(* Visualisation GAS_CALIBRATION
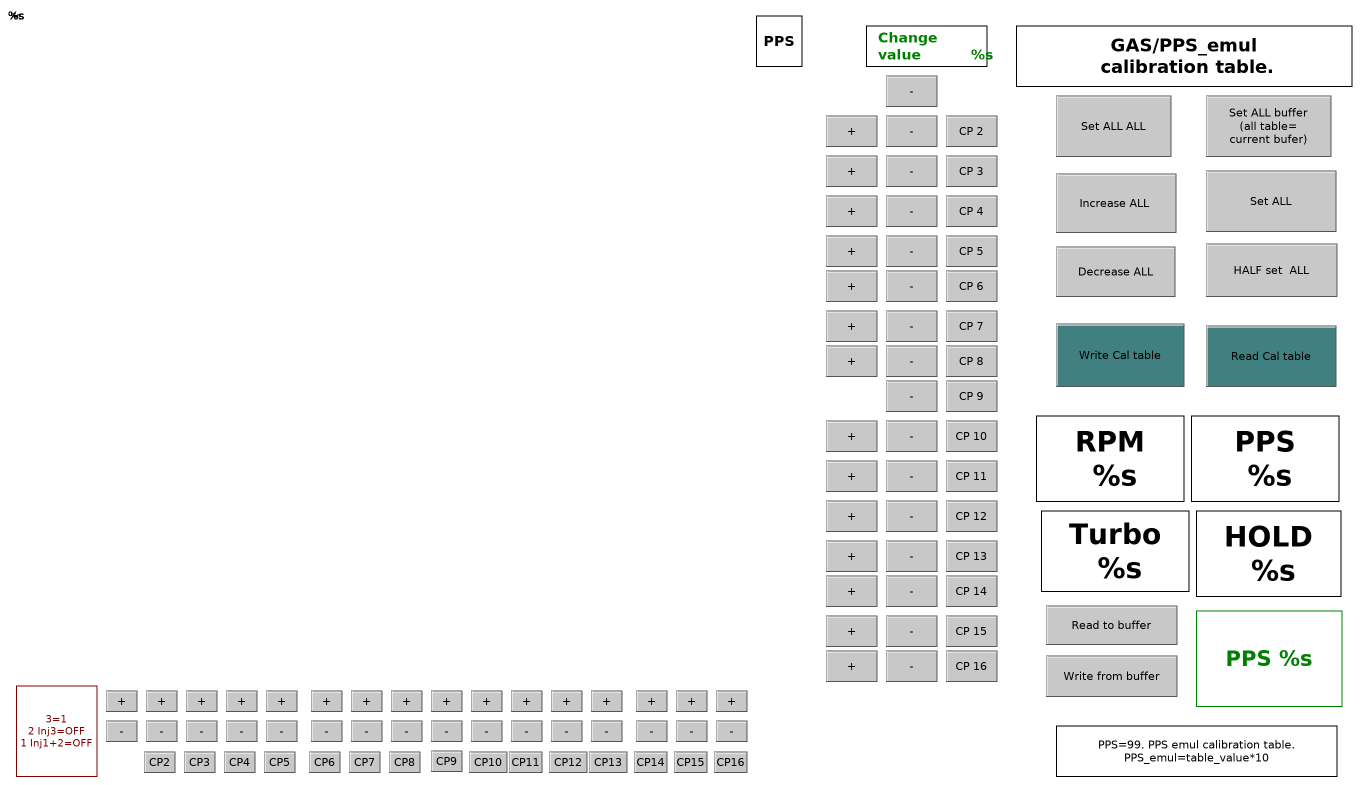
rectangle at (0,0)-(0,0): text "%s"; shows p.RPM_table[INDEX]; editable
rectangle at (0,0)-(0,0): text "%s"; shows p.Turbo_table[1]; editable
rectangle at (0,0)-(0,0): text "%s"; shows p.Turbo_table[2]; editable
rectangle at (0,0)-(0,0): text "%s"; shows p.Turbo_table[3]; editable
rectangle at (0,0)-(0,0): text "%s"; shows p.Turbo_table[4]; editable
rectangle at (0,0)-(0,0): text "%s"; shows p.Turbo_table[5]; editable
rectangle at (0,0)-(0,0): text "%s"; shows p.Turbo_table[6]; editable
rectangle at (0,0)-(0,0): text "%s"; shows p.Turbo_table[7]; editable
rectangle at (0,0)-(0,0): text "%s"; shows p.Turbo_table[8]; editable
rectangle at (0,0)-(0,0): text "%s"; shows p.Turbo_table[9]; editable
rectangle at (0,0)-(0,0): text "%s"; shows p.Turbo_table[10]; editable
rectangle at (0,0)-(0,0): text "%s"; shows p.Turbo_table[11]; editable
rectangle at (0,0)-(0,0): text "%s"; shows p.Turbo_table[12]; editable
rectangle at (0,0)-(0,0): text "%s"; shows p.Turbo_table[13]; editable
rectangle at (0,0)-(0,0): text "%s"; shows p.Turbo_table[14]; editable
rectangle at (0,0)-(0,0): text "%s"; shows p.Turbo_table[15]; editable
rectangle at (0,0)-(0,0): text "%s"; shows p.Turbo_table[16]; editable
rounded rectangle at (1180,595)-(1326,691): text "PPS %s"; shows DFPRS_Change_Cal_Table.PPS_number; editable
button at (1040,158)-(1160,217): text "Increase ALL"; taps DFPRS_Change_Cal_Table.ALL_plus
button at (1040,231)-(1159,281): text "Decrease ALL"; taps DFPRS_Change_Cal_Table.ALL_minus
button at (1190,310)-(1320,371): text "Read Cal table"; taps DFPRS_Change_Cal_Table.Read_cal
button at (1040,308)-(1168,371): text "Write Cal table"; taps DFPRS_Change_Cal_Table.Write_cal
button at (1190,155)-(1320,216): text "Set ALL"; taps DFPRS_Change_Cal_Table.Set_ALL
button at (1190,228)-(1321,281): text "HALF set  ALL"; taps DFPRS_Change_Cal_Table.HALF_set_ALL
button at (870,60)-(921,91): text "-"; taps DFPRS_Change_Cal_Table.RPM_Flag_minus_1
button at (810,100)-(861,131): text "+"; taps DFPRS_Change_Cal_Table.RPM_Flag_plus_2
button at (870,100)-(921,131): text "-"; taps DFPRS_Change_Cal_Table.RPM_Flag_minus_2
button at (930,100)-(981,131): text "CP 2"; taps DFPRS_Change_Cal_Table.RPM_Flag_CP_2
button at (810,140)-(861,171): text "+"; taps DFPRS_Change_Cal_Table.RPM_Flag_plus_3
button at (870,140)-(921,171): text "-"; taps DFPRS_Change_Cal_Table.RPM_Flag_minus_3
button at (930,140)-(981,171): text "CP 3"; taps DFPRS_Change_Cal_Table.RPM_Flag_CP_3
button at (810,180)-(861,211): text "+"; taps DFPRS_Change_Cal_Table.RPM_Flag_plus_4
button at (870,180)-(921,211): text "-"; taps DFPRS_Change_Cal_Table.RPM_Flag_minus_4
button at (930,180)-(981,211): text "CP 4"; taps DFPRS_Change_Cal_Table.RPM_Flag_CP_4
button at (810,220)-(861,251): text "+"; taps DFPRS_Change_Cal_Table.RPM_Flag_plus_5
button at (870,220)-(921,251): text "-"; taps DFPRS_Change_Cal_Table.RPM_Flag_minus_5
button at (930,220)-(981,251): text "CP 5"; taps DFPRS_Change_Cal_Table.RPM_Flag_CP_5
button at (810,255)-(861,286): text "+"; taps DFPRS_Change_Cal_Table.RPM_Flag_plus_6
button at (870,255)-(921,286): text "-"; taps DFPRS_Change_Cal_Table.RPM_Flag_minus_6
button at (930,255)-(981,286): text "CP 6"; taps DFPRS_Change_Cal_Table.RPM_Flag_CP_6
button at (810,295)-(861,326): text "+"; taps DFPRS_Change_Cal_Table.RPM_Flag_plus_7
button at (870,295)-(921,326): text "-"; taps DFPRS_Change_Cal_Table.RPM_Flag_minus_7
button at (930,295)-(981,326): text "CP 7"; taps DFPRS_Change_Cal_Table.RPM_Flag_CP_7
button at (810,330)-(861,361): text "+"; taps DFPRS_Change_Cal_Table.RPM_Flag_plus_8
button at (870,330)-(921,361): text "-"; taps DFPRS_Change_Cal_Table.RPM_Flag_minus_8
button at (930,330)-(981,361): text "CP 8"; taps DFPRS_Change_Cal_Table.RPM_Flag_CP_8
button at (90,675)-(121,696): text "+"; taps DFPRS_Change_Cal_Table.Turbo_Flag_plus_1
button at (90,705)-(121,726): text "-"; taps DFPRS_Change_Cal_Table.Turbo_Flag_minus_1
button at (130,675)-(161,696): text "+"; taps DFPRS_Change_Cal_Table.Turbo_Flag_plus_2
button at (130,705)-(161,726): text "-"; taps DFPRS_Change_Cal_Table.Turbo_Flag_minus_2
button at (128,736)-(159,757): text "CP2"; taps DFPRS_Change_Cal_Table.Turbo_Flag_CP_2
button at (170,675)-(201,696): text "+"; taps DFPRS_Change_Cal_Table.Turbo_Flag_plus_3
button at (170,705)-(201,726): text "-"; taps DFPRS_Change_Cal_Table.Turbo_Flag_minus_3
button at (168,736)-(199,757): text "CP3"; taps DFPRS_Change_Cal_Table.Turbo_Flag_CP_3
button at (210,675)-(241,696): text "+"; taps DFPRS_Change_Cal_Table.Turbo_Flag_plus_4
button at (210,705)-(241,726): text "-"; taps DFPRS_Change_Cal_Table.Turbo_Flag_minus_4
button at (208,736)-(239,757): text "CP4"; taps DFPRS_Change_Cal_Table.Turbo_Flag_CP_4
button at (250,675)-(281,696): text "+"; taps DFPRS_Change_Cal_Table.Turbo_Flag_plus_5
button at (250,705)-(281,726): text "-"; taps DFPRS_Change_Cal_Table.Turbo_Flag_minus_5
button at (248,736)-(279,757): text "CP5"; taps DFPRS_Change_Cal_Table.Turbo_Flag_CP_5
button at (295,675)-(326,696): text "+"; taps DFPRS_Change_Cal_Table.Turbo_Flag_plus_6
button at (295,705)-(326,726): text "-"; taps DFPRS_Change_Cal_Table.Turbo_Flag_minus_6
button at (293,736)-(324,757): text "CP6"; taps DFPRS_Change_Cal_Table.Turbo_Flag_CP_6
button at (335,675)-(366,696): text "+"; taps DFPRS_Change_Cal_Table.Turbo_Flag_plus_7
button at (335,705)-(366,726): text "-"; taps DFPRS_Change_Cal_Table.Turbo_Flag_minus_7
button at (333,736)-(364,757): text "CP7"; taps DFPRS_Change_Cal_Table.Turbo_Flag_CP_7
button at (375,675)-(406,696): text "+"; taps DFPRS_Change_Cal_Table.Turbo_Flag_plus_8
button at (375,705)-(406,726): text "-"; taps DFPRS_Change_Cal_Table.Turbo_Flag_minus_8
button at (373,736)-(404,757): text "CP8"; taps DFPRS_Change_Cal_Table.Turbo_Flag_CP_8
rounded rectangle at (850,10)-(971,51): text "Change / value          %s"; shows DFPRS_Change_Cal_Table.Change_volume; editable 1..
rounded rectangle at (1175,400)-(1323,486): text "PPS / %s"; shows .PPS1
rounded rectangle at (1180,495)-(1325,581): text "HOLD / %s"; shows .HOLD_time
rounded rectangle at (1000,10)-(1336,71): text "GAS/PPS_emul / calibration table."
button at (1030,590)-(1161,629): text "Read to buffer"; taps DFPRS_Change_Cal_Table.red_cal2
button at (1030,640)-(1161,681): text "Write from buffer"; taps DFPRS_Change_Cal_Table.Write_cal2
rounded rectangle at (1020,400)-(1168,486): text "RPM / %s"; shows .RPM
rounded rectangle at (1025,495)-(1173,576): text "Turbo / %s"; shows .Turbo_pressure
rounded rectangle at (740,0)-(786,51): text "PPS"
button at (870,365)-(921,396): text "-"; taps DFPRS_Change_Cal_Table.RPM_Flag_minus_9
button at (810,405)-(861,436): text "+"; taps DFPRS_Change_Cal_Table.RPM_Flag_plus_10
button at (870,405)-(921,436): text "-"; taps DFPRS_Change_Cal_Table.RPM_Flag_minus_10
button at (930,405)-(981,436): text "CP 10"; taps DFPRS_Change_Cal_Table.RPM_Flag_CP_10
button at (810,445)-(861,476): text "+"; taps DFPRS_Change_Cal_Table.RPM_Flag_plus_11
button at (870,445)-(921,476): text "-"; taps DFPRS_Change_Cal_Table.RPM_Flag_minus_11
button at (930,445)-(981,476): text "CP 11"; taps DFPRS_Change_Cal_Table.RPM_Flag_CP_11
button at (810,485)-(861,516): text "+"; taps DFPRS_Change_Cal_Table.RPM_Flag_plus_12
button at (870,485)-(921,516): text "-"; taps DFPRS_Change_Cal_Table.RPM_Flag_minus_12
button at (930,485)-(981,516): text "CP 12"; taps DFPRS_Change_Cal_Table.RPM_Flag_CP_12
button at (810,525)-(861,556): text "+"; taps DFPRS_Change_Cal_Table.RPM_Flag_plus_13
button at (870,525)-(921,556): text "-"; taps DFPRS_Change_Cal_Table.RPM_Flag_minus_13
button at (930,525)-(981,556): text "CP 13"; taps DFPRS_Change_Cal_Table.RPM_Flag_CP_13
button at (810,560)-(861,591): text "+"; taps DFPRS_Change_Cal_Table.RPM_Flag_plus_14
button at (870,560)-(921,591): text "-"; taps DFPRS_Change_Cal_Table.RPM_Flag_minus_14
button at (930,560)-(981,591): text "CP 14"; taps DFPRS_Change_Cal_Table.RPM_Flag_CP_14
button at (810,600)-(861,631): text "+"; taps DFPRS_Change_Cal_Table.RPM_Flag_plus_15
button at (870,600)-(921,631): text "-"; taps DFPRS_Change_Cal_Table.RPM_Flag_minus_15
button at (930,600)-(981,631): text "CP 15"; taps DFPRS_Change_Cal_Table.RPM_Flag_CP_15
button at (810,635)-(861,666): text "+"; taps DFPRS_Change_Cal_Table.RPM_Flag_plus_16
button at (870,635)-(921,666): text "-"; taps DFPRS_Change_Cal_Table.RPM_Flag_minus_16
button at (930,635)-(981,666): text "CP 16"; taps DFPRS_Change_Cal_Table.RPM_Flag_CP_16
button at (930,365)-(981,396): text "CP 9"; taps DFPRS_Change_Cal_Table.RPM_Flag_CP_9
button at (415,675)-(446,696): text "+"; taps DFPRS_Change_Cal_Table.Turbo_Flag_plus_9
button at (415,705)-(446,726): text "-"; taps DFPRS_Change_Cal_Table.Turbo_Flag_minus_9
button at (455,675)-(486,696): text "+"; taps DFPRS_Change_Cal_Table.Turbo_Flag_plus_10
button at (455,705)-(486,726): text "-"; taps DFPRS_Change_Cal_Table.Turbo_Flag_minus_10
button at (453,736)-(491,757): text "CP10"; taps DFPRS_Change_Cal_Table.Turbo_Flag_CP_10
button at (495,675)-(526,696): text "+"; taps DFPRS_Change_Cal_Table.Turbo_Flag_plus_11
button at (495,705)-(526,726): text "-"; taps DFPRS_Change_Cal_Table.Turbo_Flag_minus_11
button at (493,736)-(526,757): text "CP11"; taps DFPRS_Change_Cal_Table.Turbo_Flag_CP_11
button at (535,675)-(566,696): text "+"; taps DFPRS_Change_Cal_Table.Turbo_Flag_plus_12
button at (535,705)-(566,726): text "-"; taps DFPRS_Change_Cal_Table.Turbo_Flag_minus_12
button at (533,736)-(571,757): text "CP12"; taps DFPRS_Change_Cal_Table.Turbo_Flag_CP_12
button at (575,675)-(606,696): text "+"; taps DFPRS_Change_Cal_Table.Turbo_Flag_plus_13
button at (575,705)-(606,726): text "-"; taps DFPRS_Change_Cal_Table.Turbo_Flag_minus_13
button at (573,736)-(611,757): text "CP13"; taps DFPRS_Change_Cal_Table.Turbo_Flag_CP_13
button at (620,675)-(651,696): text "+"; taps DFPRS_Change_Cal_Table.Turbo_Flag_plus_14
button at (620,705)-(651,726): text "-"; taps DFPRS_Change_Cal_Table.Turbo_Flag_minus_14
button at (618,736)-(651,757): text "CP14"; taps DFPRS_Change_Cal_Table.Turbo_Flag_CP_14
button at (660,675)-(691,696): text "+"; taps DFPRS_Change_Cal_Table.Turbo_Flag_plus_15
button at (660,705)-(691,726): text "-"; taps DFPRS_Change_Cal_Table.Turbo_Flag_minus_15
button at (658,736)-(691,757): text "CP15"; taps DFPRS_Change_Cal_Table.Turbo_Flag_CP_15
button at (700,675)-(731,696): text "+"; taps DFPRS_Change_Cal_Table.Turbo_Flag_plus_16
button at (700,705)-(731,726): text "-"; taps DFPRS_Change_Cal_Table.Turbo_Flag_minus_16
button at (698,736)-(731,757): text "CP16"; taps DFPRS_Change_Cal_Table.Turbo_Flag_CP_16
button at (415,735)-(446,756): text "CP9"; taps DFPRS_Change_Cal_Table.Turbo_Flag_CP_9
button at (1040,80)-(1155,141): text "Set ALL ALL"; taps DFPRS_Change_Cal_Table.Set_ALL_ALL
button at (1190,80)-(1315,141): text "Set ALL buffer / (all table= / current bufer)"; taps DFPRS_Change_Cal_Table.Set_ALL_ALL
rectangle at (0,670)-(81,761): text "3=1 / 2 Inj3=OFF / 1 Inj1+2=OFF"
rectangle at (0,0)-(0,0): text "%s"; shows p.PPS_table[INDEX]; editable
rectangle at (1040,710)-(1321,761): text "PPS=99. PPS emul calibration table. / PPS_emul=table_value*10"
*)

(* Visualisation MAIN_PRIBOR
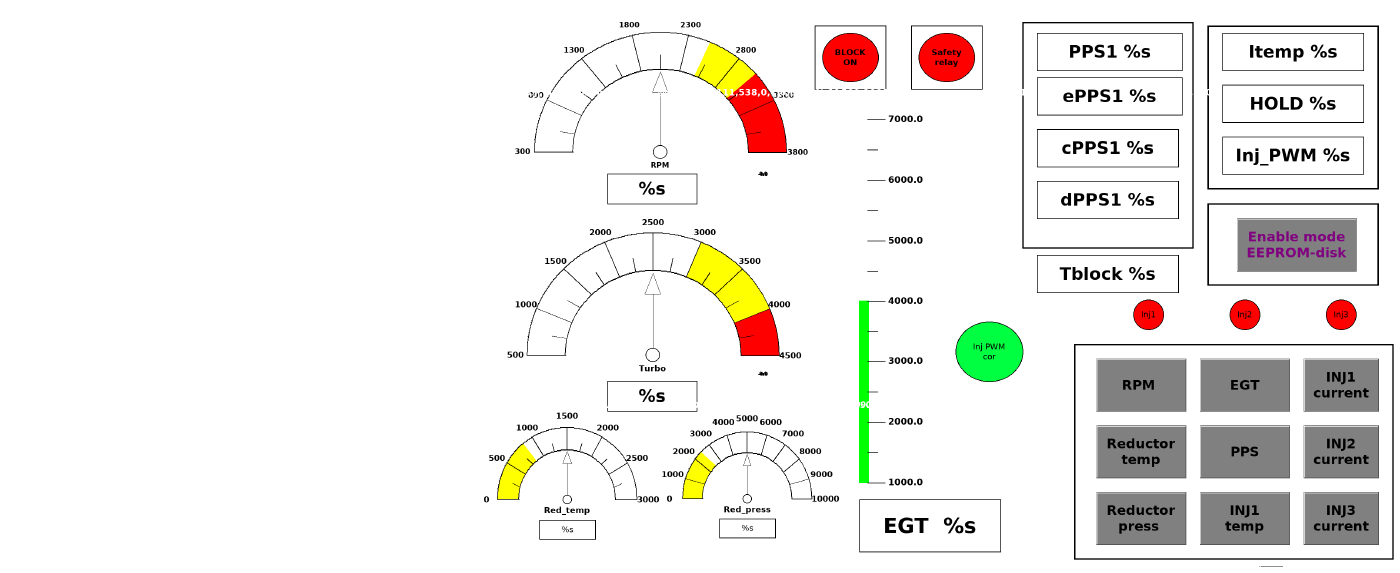
group at (60,0)-(461,216)
  rectangle at (0,0)-(1,1): text "{ExtendedElement},Visu\ElementDLL.ete,0,@Zeigerinstrument,401,180,0,0,255,255,255,0,RPM,RPM,%.0f,0,1,1,250,500,300,3800,0,0,0,0,0,0,0,-13,16,700,Arial,1,2,3000,3800,255,0,0,2500,2999,255,255,0,"
  rectangle at (5,192)-(26,208): text "300"
  rectangle at (23,112)-(44,128): text "800"
  rectangle at (71,48)-(99,64): text "1300"
  rectangle at (145,12)-(173,28): text "1800"
  rectangle at (228,12)-(256,28): text "2300"
  rectangle at (302,48)-(330,64): text "2800"
  rectangle at (353,112)-(381,128): text "3300"
  rectangle at (372,193)-(400,209): text "3800"
  rectangle at (186,211)-(215,227): text "RPM"
  polygon at (190,87)-(211,201): angle ((RPM * 1.0)-2050) * 0.0514286
group at (400,220)-(401,221)
  rectangle at (0,0)-(1,1): text "{ExtendedElement},Visu\ElementDLL.ete,0,@Zeigerinstrument,200,180,0,0,255,255,255,0,,,%.1f,0,1,1,1,2,-4,4,0,0,0,0,0,0,0,-13,16,700,Arial,1,2,4000,5500,255,255,128,5500,6000,255,0,0,"
  rectangle at (1,92)-(23,108): text "-4.0"
  rectangle at (27,30)-(49,46): text "-2.0"
  rectangle at (91,4)-(109,20): text "0.0"
  rectangle at (153,30)-(171,46): text "2.0"
  rectangle at (179,92)-(197,108): text "4.0"
group at (400,490)-(401,491)
  rectangle at (0,0)-(1,1): text "{ExtendedElement},Visu\ElementDLL.ete,0,@Zeigerinstrument,200,180,0,0,255,255,255,0,,,%.1f,0,1,1,1,2,-4,4,0,0,0,0,0,0,0,-13,16,700,Arial,1,2,4000,5500,255,255,128,5500,6000,255,0,0,"
  rectangle at (1,92)-(23,108): text "-4.0"
  rectangle at (27,30)-(49,46): text "-2.0"
  rectangle at (91,4)-(109,20): text "0.0"
  rectangle at (153,30)-(171,46): text "2.0"
  rectangle at (179,92)-(197,108): text "4.0"
group at (50,270)-(451,491)
  rectangle at (0,0)-(1,1): text "{ExtendedElement},Visu\ElementDLL.ete,0,@Zeigerinstrument,401,180,0,0,255,255,255,0,Turbo_pressure,Turbo,%.0f,0,1,1,250,500,500,4500,0,0,0,0,0,0,0,-13,16,700,Arial,1,2,3000,4000,255,255,0,4000,4500,255,0,0,"
  rectangle at (5,192)-(26,208): text "500"
  rectangle at (16,122)-(44,138): text "1000"
  rectangle at (56,62)-(84,78): text "1500"
  rectangle at (116,22)-(144,38): text "2000"
  rectangle at (187,8)-(215,24): text "2500"
  rectangle at (257,22)-(285,38): text "3000"
  rectangle at (317,62)-(345,78): text "3500"
  rectangle at (357,122)-(385,138): text "4000"
  rectangle at (372,193)-(400,209): text "4500"
  rectangle at (182,211)-(219,227): text "Turbo"
  polygon at (190,87)-(211,201): angle ((Turbo_pressure * 1.0)-2500) * 0.045
rounded rectangle at (190,500)-(311,541): text "%s"; shows .Turbo_pressure
rounded rectangle at (190,220)-(311,261): text "%s"; shows .RPM
group at (510,110)-(621,648)
  rectangle at (0,0)-(1,1): text "{ExtendedElement},Visu\ElementDLL.ete,1,@Bargraph,111,538,0,1,0,EGT,,%.1f,500,1000,1000,7000,0,0,0,0,0,0,0,-13,16,700,Arial,0,255,0,255,0,0,1,6000,0,0,0,"
  rectangle at (18,268)-(30,502): alarm colour if (EGT) > 6000; top ((EGT * 1.0) - 4000)  * -0.078
  rectangle at (53,491)-(103,512): text "1000.0"
  rectangle at (53,413)-(103,434): text "2000.0"
  rectangle at (53,335)-(103,356): text "3000.0"
  rectangle at (53,258)-(103,279): text "4000.0"
  rectangle at (53,180)-(103,201): text "5000.0"
  rectangle at (53,102)-(103,123): text "6000.0"
  rectangle at (53,24)-(103,45): text "7000.0"
group at (11,532)-(259,683)
  rectangle at (0,0)-(1,1): text "{ExtendedElement},Visu\ElementDLL.ete,0,@Zeigerinstrument,248,180,0,0,255,255,255,0,Reductor_temp,Red_temp,%.0f,0,1,1,250,500,0,3000,0,0,0,0,0,0,0,-13,16,700,Arial,1,1,0,850,255,255,0,"
  rectangle at (12,116)-(19,132): text "0"
  rectangle at (19,62)-(40,78): text "500"
  rectangle at (56,22)-(84,38): text "1000"
  rectangle at (110,7)-(138,23): text "1500"
  rectangle at (165,22)-(193,38): text "2000"
  rectangle at (204,62)-(232,78): text "2500"
  rectangle at (219,116)-(247,132): text "3000"
  rectangle at (92,130)-(156,146): text "Red_temp"
  polygon at (118,61)-(130,124): angle ((Reductor_temp * 1.0)-1500) * 0.06
rounded rectangle at (98,688)-(174,714): text "%s"; shows .Reductor_temp
rounded rectangle at (530,660)-(721,731): text "EGT  %s"; shows .EGT
ellipse at (480,30)-(556,96): text "BLOCK / ON"; alarm colour if .Flag_ECU_ON
rounded rectangle at (1020,100)-(1211,151): text "HOLD %s"; shows .HOLD_time
group at (254,531)-(502,682)
  rectangle at (0,0)-(1,1): text "{ExtendedElement},Visu\ElementDLL.ete,0,@Zeigerinstrument,248,180,0,0,255,255,255,0,Reductor_press,Red_press,%.0f,0,1,1,1000,1000,0,10000,0,0,0,0,0,0,0,-13,16,700,Arial,1,1,0,2500,255,255,0,"
  rectangle at (16,116)-(23,132): text "0"
  rectangle at (10,84)-(38,100): text "1000"
  rectangle at (25,54)-(53,70): text "2000"
  rectangle at (48,31)-(76,47): text "3000"
  rectangle at (78,16)-(106,32): text "4000"
  rectangle at (110,11)-(138,27): text "5000"
  rectangle at (142,16)-(170,32): text "6000"
  rectangle at (172,31)-(200,47): text "7000"
  rectangle at (195,54)-(223,70): text "8000"
  rectangle at (210,84)-(238,100): text "9000"
  rectangle at (212,116)-(247,132): text "10000"
  rectangle at (92,130)-(157,146): text "Red_press"
  polygon at (119,66)-(129,124): angle ((Reductor_press * 1.0)-5000) * 0.018
rounded rectangle at (341,686)-(417,712): text "%s"; shows .Reductor_press
rounded rectangle at (1020,30)-(1211,81): text "Itemp %s"; shows .Injector_temp
rounded rectangle at (770,30)-(966,81): text "PPS1 %s"; shows .PPS1
rounded rectangle at (770,90)-(966,141): text "ePPS1 %s"; shows .PPS1_emul
button at (850,470)-(971,541): text "RPM"; toggles .Err_RPM
button at (990,470)-(1111,541): text "EGT"; toggles .Err_EGT
button at (850,560)-(971,631): text "Reductor / temp"; toggles .Err_Reductor_temp
button at (850,650)-(971,721): text "Reductor / press"; shows .Reductor_press; toggles .Err_Reductor_press
button at (1130,470)-(1231,541): text "INJ1 / current"; toggles .Err_Inj1
button at (1130,560)-(1231,631): text "INJ2 / current"; toggles .Err_Inj2
button at (990,650)-(1111,721): text "INJ1 / temp"; toggles .Err_Inj_temp
button at (990,560)-(1111,631): text "PPS"; toggles .Err_PPS
button at (1040,280)-(1201,352): text "Enable mode / EEPROM-disk"; toggles .Flag_CAN
button at (1130,650)-(1231,721): text "INJ3 / current"; toggles .Err_Inj3
rounded rectangle at (770,330)-(961,381): text "Tblock %s"; shows .gs16_TempBoard
ellipse at (900,390)-(941,431): text "Inj1"; alarm colour if .Flag_Inj1_ON
ellipse at (1030,390)-(1071,431): text "Inj2"; alarm colour if .Flag_Inj2_ON
ellipse at (1160,390)-(1201,431): text "Inj3"; alarm colour if .Flag_Inj3_ON
ellipse at (610,30)-(686,96): text "Safety / relay"; alarm colour if .gq_Relay
rounded rectangle at (770,160)-(961,211): text "cPPS1 %s"; shows .cPPS1_emul
rounded rectangle at (1020,170)-(1211,221): text "Inj_PWM %s"; shows .Inj_PWM_time
rounded rectangle at (770,230)-(961,281): text "dPPS1 %s"; shows .PPS1-.cPPS1_emul
ellipse at (660,420)-(751,501): text "Inj PWM / cor"; alarm colour if .Flag_Inj_PWM_cor
120 more shapes without text or variables
*)

(* Visualisation PLC_VISU
1 more shapes without text or variables
*)

(* Visualisation PWM_ADJUSTMENT
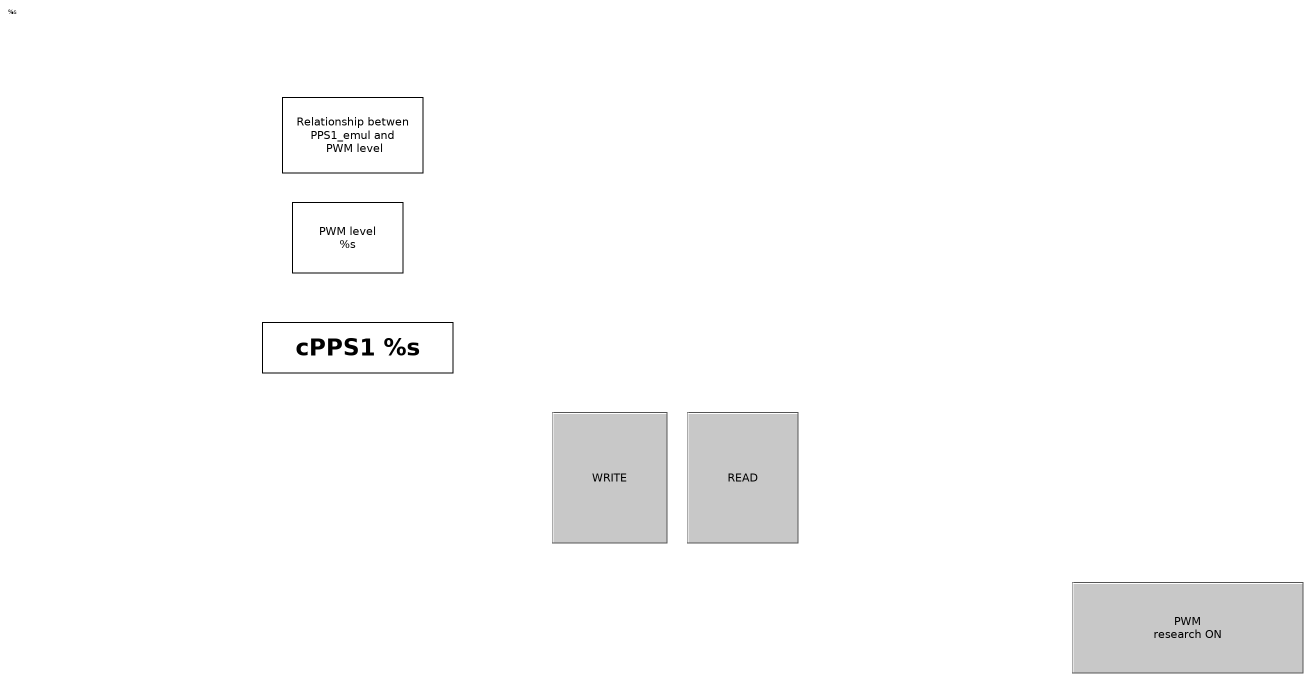
button at (1060,570)-(1291,661): text "PWM / research ON"; toggles .Flag_PWM_researh
button at (540,400)-(655,531): text "WRITE"; taps DFPRS_Change_Cal_Table.Write_cal
button at (675,400)-(786,531): text "READ"; taps DFPRS_Change_Cal_Table.Read_cal
rounded rectangle at (270,85)-(411,161): text "Relationship betwen / PPS1_emul and / PWM level"
rounded rectangle at (280,190)-(391,261): text "PWM level / %s"; shows Act_control.j; editable
rectangle at (0,0)-(0,0): text "%s"; shows p.PPS1_emul_PWM[INDEX]; editable
rounded rectangle at (250,310)-(441,361): text "cPPS1 %s"; shows .cPPS1_emul
1 elements of other kinds (tables, trends, ...) not read
*)
